FUNCTION_BLOCK XtsMover IMPLEMENTS I_Cyclic, I_XtsMover, I_Resettable, I_Object
VAR
	MyAxisRef : AXIS_REF;
	_MyAxisStatus : ST_AxisStatus;
	_MyNCData : NCTOPLC_AXIS_REF;
	TaskCollection : ObjectRunner<99>;
	EnableBehaviour : EnableDisableTask := (AxisRef := MyAxisRef);
	MoveBehaviour : MoveToPositionTask:= (AxisRef := MyAxisRef);
	HaltBehaviour : HaltMoverTask := (AxisRef := MyAxisRef);
	ResetBehaviour : CoEResetTask := (AxisRef := MyAxisRef);
	MoverActivateTrackBehaviour : ActivateTrackTask:= (AxisRef := MyAxisRef);
	_ipTcIoXtsMover	: I_TcIoXtsXpuMover;
	TrackChangeTrigger : R_TRIG;
	_MoverAbsMoveOptions : ST_MoveAbsoluteCAOptions;
	_stTmsActPositions : ST_PositionInfo;
	_CurrentTrack : I_XtsTrack;
	_myStatus : MoverStatus;
	_MyCAGroup : I_CollisionGroup;
	_ForwardOnly : BOOL := TRUE;
	myControllerOid: OTCID;
	MyId: UDINT;
	MoverID : T_MaxString;
	Initialised : BOOL;
	MyTrackCount : INT;
	MyTracks : ARRAY[0..MaxTracks] OF I_XtsTrack;
	NullTrack : XtsTrack('');
	_SetForce: LREAL;
	_SetCurrent: LREAL;
	_Gap : LREAL;
	_Acceleration : LREAL;
	_Deceleration : LREAL;
	_Jerk : LREAL;
	_DistanceDrivenInMM : LREAL;
	_AvoidingCollision: BOOL;
	_Mover1 : BOOL;
	myController: Tc3_XTS_Utility.I_McXtsMoverController;
END_VAR
VAR CONSTANT
	_MaxMoverVelocity : MC_LREAL := 4000.0;
	MaxTracks : INT := 5;
	InPositionToleranceForMoveChecks : LREAL := 0.001;
END_VAR

PROPERTY PUBLIC Acceleration : MC_LREAL
GET
Acceleration := MoveBehaviour.Acceleration;
END_GET
SET
MoveBehaviour.Acceleration := Acceleration;
_Acceleration := Acceleration;
END_SET
END_PROPERTY

METHOD ActivateTrack : HRESULT
VAR_INPUT
	Track : INT;
END_VAR
IF Track = 0 THEN
	ActivateTrack := -1;
	Base_Library.Tracing.Trace.Warning(MoverID, 'ActivateTrack Fail - Null Track');
	RETURN;
END_IF
IF MoverActivateTrackBehaviour.Busy THEN
	ActivateTrack := -2;
	Base_Library.Tracing.Trace.Warning(MoverID, 'ActivateTrack Fail - Activating');
	RETURN;
END_IF

IF NOT THIS^.IsStationary THEN
	ActivateTrack := -3;
	Base_Library.Tracing.Trace.Warning(MoverID, 'ActivateTrack Fail - Moving');
	RETURN;
END_IF

IF Track > MyTrackCount THEN
	ActivateTrack := -4;
	Base_Library.Tracing.Trace.Warning(MoverID, 'ActivateTrack Fail - Track not Registered');
	RETURN;
END_IF

IF MyTracks[Track - 1].MyOTCID = 0  THEN
	ActivateTrack := -5;
	Base_Library.Tracing.Trace.Warning(MoverID, 'ActivateTrack Fail - No Track');
	RETURN;
END_IF
	
Base_Library.Tracing.Trace.Verbose(MoverID, 'ActivateTrack Request Accepted');
MoverActivateTrackBehaviour.Execute(Track := MyTracks[Track - 1]);
_ipTcIoXtsMover.SetActiveTrackObjectId(nTrackObjectId := MyTracks[Track - 1].MyOTCID);
_CurrentTrack := MyTracks[Track - 1];
END_METHOD

METHOD ActivateZeroReferenceSystem : HRESULT
IF MoverActivateTrackBehaviour.Busy THEN
	ActivateZeroReferenceSystem := -1;
	Base_Library.Tracing.Trace.Warning(MoverID, 'ActivateZeroTrack Fail - Activating');
	RETURN;
END_IF
IF NOT THIS^.IsStationary THEN
	ActivateZeroReferenceSystem := -2;
	Base_Library.Tracing.Trace.Warning(MoverID, 'ActivateZeroTrack Fail - Moving');
	RETURN;
END_IF 

Base_Library.Tracing.Trace.Verbose(MoverID, 'ActivateTrack Request Accpeted');
MoverActivateTrackBehaviour.Execute(Track := NullTrack);
_CurrentTrack := 0;
END_METHOD

PROPERTY ActualForce : LREAL
GET
ActualForce := _SetForce;
END_GET
END_PROPERTY

PROPERTY ActualPosition : LREAL
GET
ActualPosition := MyAxisRef.NcToPlc.ActPos;
END_GET
END_PROPERTY

PROPERTY ActualTrackPosition : LREAL
GET
ActualTrackPosition := _stTmsActPositions.fTrackPosition;
END_GET
END_PROPERTY

PROPERTY ActualVelocity : LREAL
GET
ActualVelocity := MyAxisRef.NcToPlc.ActVelo;
END_GET
END_PROPERTY

PROPERTY AxisRef : Reference to Axis_ref
GET
AxisRef REF= MyAxisRef;
END_GET
END_PROPERTY

METHOD PUBLIC  Cycle : HRESULT
VAR_INPUT
END_VAR
IF Initialised THEN
	TaskCollection.Cycle();
	TrackChangeTrigger(CLK := MoverActivateTrackBehaviour.Done);
	IF TrackChangeTrigger.Q THEN
		_MoverAbsMoveOptions.PositionReferenceSystem :=  MoverActivateTrackBehaviour.NewTrackId;
		_MoverAbsMoveOptions.DynamicsReferenceSystem := MoverActivateTrackBehaviour.NewTrackId;
		MoveBehaviour.Options := _MoverAbsMoveOptions;	
	END_IF
	IF _ipTcIoXtsMover <> 0 THEN
		_stTmsActPositions := _ipTcIoXtsMover.GetPositionInfo();
		_SetForce := _ipTcIoXtsMover.GetSetForce();
		_SetCurrent := _ipTcIoXtsMover.GetSetCurrent();
		_myStatus.isMover1 := _ipTcIoXtsMover.GetIsMover1();
		_myStatus.isActive := _ipTcIoXtsMover.GetIsActive();
		_myStatus.isFrozen := _ipTcIoXtsMover.GetIsFrozen();
		_myStatus.isLost := _ipTcIoXtsMover.GetIsLost();
		_myStatus.isReadyForPositioning := _ipTcIoXtsMover.GetIsReadyForPositioning();
		_myStatus.hasControllerError := _ipTcIoXtsMover.GetMoverControllerError();
		_myStatus.driveState := _ipTcIoXtsMover.GetDriveStatus();
		_DistanceDrivenInMM := _ipTcIoXtsMover.GetDistanceDriven();
	END_IF
	_AvoidingCollision := MyAxisRef.NcToPlc.StateDWord2.Flags.AvoidingCollision;
ELSE
	Cycle := -1;
END_IF
MyAxisRef.ReadStatus();
_MyNCData := MyAxisRef.NcToPlc;
_MyAxisStatus := MyAxisRef.Status;
END_METHOD

PROPERTY PUBLIC Deceleration : MC_LREAL
GET
Deceleration := MoveBehaviour.Deceleration;
END_GET
SET
MoveBehaviour.Deceleration := Deceleration;
HaltBehaviour.Deceleration := Deceleration;
_Deceleration := Deceleration;
END_SET
END_PROPERTY

METHOD PUBLIC DisableMover : HRESULT
VAR_INPUT
END_VAR
IF NOT THIS^.IsEnabled THEN
	DisableMover := -1;
	Base_Library.Tracing.Trace.Warning(MoverID, 'Disable request Fail - Disabled'); 
	RETURN;
END_IF
	
Base_Library.Tracing.Trace.Verbose(MoverID, 'Disable Request Accepted');
EnableBehaviour.Disable();
END_METHOD

METHOD PUBLIC EnableMover : HRESULT
VAR_INPUT
END_VAR
IF EnableBehaviour.Busy THEN
	EnableMover := -1;
	Base_Library.Tracing.Trace.Warning(MoverID, 'Enable Request Failed - Enabling');
	RETURN;
END_IF
IF THIS^.IsEnabled THEN
	EnableMover := -2;
	Base_Library.Tracing.Trace.Warning(MoverID, 'Enable Request Failed - Enabled');
	RETURN;
END_IF
	
Base_Library.Tracing.Trace.Verbose(MoverID, 'Enable Request Accepted');
EnableBehaviour.Enable();
END_METHOD

PROPERTY ErrorID : UDINT
GET
ErrorID := _MyAxisStatus.ErrorID;
END_GET
END_PROPERTY

//FB_Init is always available implicitly and it is used primarily for initialization.
//The return value is not evaluated. For a specific influence, you can also declare the
//methods explicitly and provide additional code there with the standard initialization
//code. You can evaluate the return value.
METHOD FB_Init: BOOL
VAR_INPUT
    bInitRetains: BOOL; // TRUE: the retain variables are initialized (reset warm / reset cold)
    bInCopyCode: BOOL;  // TRUE: the instance will be copied to the copy code afterward (online change)   
END_VAR
TaskCollection.RegisterCyclic(EnableBehaviour);
TaskCollection.RegisterCyclic(ResetBehaviour);
TaskCollection.RegisterCyclic(HaltBehaviour);
TaskCollection.RegisterCyclic(MoveBehaviour);
TaskCollection.RegisterCyclic(MoverActivateTrackBehaviour);
END_METHOD

PROPERTY PUBLIC Gap : MC_LREAL
GET
Gap := MoveBehaviour.Gap;
END_GET
SET
IF Gap >= 50.0 THEN
	MoveBehaviour.Gap := Gap;
	HaltBehaviour.Gap := Gap;
	_Gap := Gap;
ELSE
	_Gap := 100.0;
	MoveBehaviour.Gap := 100.0;
	HaltBehaviour.Gap := 100.0;
END_IF
END_SET
END_PROPERTY

METHOD GetActiveTrackLength : LREAL
VAR_INPUT
END_VAR
GetActiveTrackLength := _CurrentTrack.TrackLength;
END_METHOD

METHOD GetMoverCtrlOTCID : XtsMoverControllerOTCID
VAR_INPUT
END_VAR
GetMoverCtrlOTCID := _ipTcIoXtsMover.GetMoverControllerOid();
END_METHOD

METHOD GetMoverOTCID : OTCID
VAR_INPUT
END_VAR
//GetMoverCtrlOTCID := _ipTcIoXtsMover.P_AxisOid;
END_METHOD

METHOD PUBLIC HaltAxis : HRESULT
VAR_INPUT
END_VAR
IF HaltBehaviour.Busy THEN
	HaltAxis := -1;
	Base_Library.Tracing.Trace.Warning(MoverID, 'Halt Request Fail - Halting');
	RETURN;
END_IF
	
Base_Library.Tracing.Trace.Verbose(MoverID, 'Halt Request Accepted');
HaltBehaviour.Execute();
END_METHOD

PROPERTY HasError : BOOL
GET
HasError := _MyAxisStatus.Error;
END_GET
END_PROPERTY

PROPERTY PUBLIC IdentInGroup : IDENT_IN_GROUP_REF
GET
IdentInGroup := UDINT_TO_IDENTINGROUP(id := _MyNCData.AxisId);
END_GET
END_PROPERTY

METHOD Initialise : HRESULT
VAR_INPUT
END_VAR
VAR
	i : INT;
END_VAR
IF Initialised THEN
	Initialise := -1;
	RETURN;
END_IF
IF _ipTcIoXtsMover = 0 THEN
	Initialise := -2;
	RETURN;
END_IF
IF NOT IsDetected THEN
	Initialise := -3;
	RETURN;
END_IF
IF MyTrackCount = 0 THEN
	Initialise := -4;
	RETURN;
END_IF
myController := _ipTcIoXtsMover.MoverController;
myControllerOid := _ipTcIoXtsMover.GetMoverControllerOid();
MyId := _ipTcIoXtsMover.P_AxisId;
MoverID := CONCAT('Mover ', TO_STRING(MyId));
_Mover1 := _ipTcIoXtsMover.GetIsMover1();
_CurrentTrack := MyTracks[MoversActiveTrack - 1];
Initialised := TRUE;
END_METHOD

PROPERTY IsActive : BOOL
GET
IsActive := _myStatus.isActive;
END_GET
END_PROPERTY

PROPERTY IsAMover1 : BOOL
GET
IsAMover1 := _Mover1;
END_GET
END_PROPERTY

PROPERTY IsAvoidingCollision : BOOL
GET
isAvoidingCollision := _AvoidingCollision;
END_GET
END_PROPERTY

PROPERTY IsDetected : BOOL
GET
IsDetected := MyAxisRef.NcToPlc.AxisId <> 0;
END_GET
END_PROPERTY

PROPERTY IsEnabled : BOOL
GET
IsEnabled :=  NOT _MyAxisStatus.Disabled;
END_GET
END_PROPERTY

PROPERTY IsStationary : BOOL
GET
IsStationary := _MyAxisStatus.NotMoving;
END_GET
END_PROPERTY

PROPERTY PUBLIC Jerk : MC_LREAL
GET
Jerk := MoveBehaviour.Jerk;
END_GET
SET
MoveBehaviour.Jerk := Jerk;
HaltBehaviour.Jerk := Jerk;
_Jerk := Jerk;
END_SET
END_PROPERTY

PROPERTY PUBLIC MoversActiveTrack : INT
GET
VAR
	i : INT;
END_VAR
FOR i := 0 TO MyTrackCount - 1 DO
	IF MyTracks[i].MyOTCID =  _ipTcIoXtsMover.GetActiveTrackObjectId() THEN
		MoversActiveTrack := i + 1;
		EXIT;
	END_IF
END_FOR
END_GET
END_PROPERTY

PROPERTY PUBLIC MoverXtsIoEnvInterface : I_TcIoXtsXpuMover
GET
MoverXtsIoEnvInterface := _ipTcIoXtsMover;
END_GET
SET
_ipTcIoXtsMover := MoverXtsIoEnvInterface;
END_SET
END_PROPERTY

METHOD PUBLIC MoveTo : HRESULT
VAR_INPUT
	RequiredPosition : MC_LREAL;
	MoveVelocity : MC_LREAL;
	NonModuloMove : BOOL;
END_VAR
IF MoveBehaviour.Busy THEN
	Base_Library.Tracing.Trace.Warning(MoverID, 'Mover Called While Busy');
	MoveTo := -1;
	RETURN;
END_IF
IF MoveVelocity > _MaxMoverVelocity THEN
	Base_Library.Tracing.Trace.Warning(MoverID, 'Move Velo Too High');
	MoveTo := -2;
	RETURN;
END_IF
IF MoveVelocity <= 0.0 THEN
	Base_Library.Tracing.Trace.Warning(MoverID, 'Move Velo Less Than Zero');
	MoveTo := -3;
	RETURN;
END_IF
IF Gap <= 50.0 THEN
	Base_Library.Tracing.Trace.Warning(MoverID, 'Move Gasp Too Small');
	MoveTo := -4;
	RETURN;
END_IF

Base_Library.Tracing.Trace.Verbose(moverID, concat('Move Accepted to : ',TO_STRING(RequiredPosition)));

IF NonModuloMove THEN
	THIS^.MoveBehaviour.MoveTo(Position := RequiredPosition, 
									Velocity := MoveVelocity, 
									Direction := Tc3_Mc3Definitions.MC_DIRECTION.mcDirectionNonModulo, 
									Turns := 0);
	MoveTo := 1;
END_IF

IF NOT NonModuloMove AND _ForwardOnly THEN
	MoveTo := THIS^.MoveBehaviour.MoveTo(Position := RequiredPosition, 
									Velocity := MoveVelocity, 
									Direction := Tc3_Mc3Definitions.MC_DIRECTION.mcDirectionPositive, 
									Turns := 0);
	MoveTo := 2;
END_IF

IF NOT NonModuloMove AND NOT _ForwardOnly THEN
	IF RequiredPosition > MyAxisRef.NcToPlc.ModuloActPos THEN
		MoveTo := THIS^.MoveBehaviour.MoveTo(Position := RequiredPosition, 
									Velocity := MoveVelocity, 
									Direction := Tc3_Mc3Definitions.MC_DIRECTION.mcDirectionPositive, 
									Turns := 0);
		MoveTo := 3;
	ELSE
		MoveTo := THIS^.MoveBehaviour.MoveTo(Position := RequiredPosition, 
									Velocity := MoveVelocity, 
									Direction := Tc3_Mc3Definitions.MC_DIRECTION.mcDirectionNegative, 
									Turns := 0);
		MoveTo := 4;
	END_IF
END_IF
END_METHOD

PROPERTY MyCAGroup : I_CollisionGroup
GET
MyCAGroup := _MyCAGroup;
END_GET
SET
_MyCAGroup := MyCAGroup;
END_SET
END_PROPERTY

PROPERTY PositiveDirectionOnly : BOOL
GET
PositiveDirectionOnly := _ForwardOnly;
END_GET
SET
_ForwardOnly := PositiveDirectionOnly;
END_SET
END_PROPERTY

METHOD RegisterTracks : HRESULT
VAR_INPUT
	Track : I_XtsTrack;
END_VAR
VAR
	Registered : BOOL;
	i : INT;
END_VAR
IF Track = 0 THEN
	RegisterTracks := -1;
	RETURN;
END_IF
Registered := FALSE;
FOR i := 0 TO 5 DO 
	IF Track = MyTracks[i] THEN
		Registered := TRUE;
	END_IF
END_FOR
IF Registered THEN
	RegisterTracks := -2;
	RETURN;
END_IF
FOR i := 0 TO 5 DO
	IF MyTracks[i] = 0 THEN
		MyTracks[i] := Track;
		MyTrackCount := MyTrackCount + 1;
		EXIT;
	END_IF
END_FOR
END_METHOD

METHOD RegisterWithParent
VAR_INPUT
	Parent	: I_HostObjects;
END_VAR
Parent.RegisterCyclic(THIS^);
END_METHOD

METHOD PUBLIC Reset : HRESULT
VAR_INPUT
END_VAR
IF ResetBehaviour.Busy THEN
	Base_Library.Tracing.Trace.Warning(MoverID, 'Reset Request Failed - Reseting');
	Reset := -1;
	RETURN;
END_IF
 
IF NOT (_MyAxisStatus.Error OR _MyAxisStatus.NotMoving) THEN
	Base_Library.Tracing.Trace.Warning(MoverID, 'Reset Request Failed - Not Allowed');
	Reset := -2;
	RETURN;
END_IF

Base_Library.Tracing.Trace.Verbose(MoverID, 'Reset Request Accepted');
ResetBehaviour.Reset();
MoveBehaviour.Abort();
END_METHOD

METHOD SetForceCouple : HRESULT
VAR_INPUT
	XtsMoverCtrlOTCID : Tc3_XTS_Utility.XtsMoverControllerOTCID;
END_VAR
IF _ipTcIoXtsMover = 0 THEN
	SetForceCouple := - 1;
	RETURN;
END_IF

_ipTcIoXtsMover.MoverController.SetForceCouple(nForceCouple := XtsMoverCtrlOTCID);
END_METHOD

METHOD SetMoverActiveTrack : HRESULT
VAR_INPUT
	Track : INT;
END_VAR
IF Track = 0 THEN
	SetMoverActiveTrack := -1;
	RETURN;
END_IF

IF NOT THIS^.IsStationary THEN
	SetMoverActiveTrack := -3;
	RETURN;
END_IF

IF Track > MyTrackCount THEN
	SetMoverActiveTrack := -4;
	RETURN;
END_IF

IF MyTracks[Track - 1].MyOTCID = 0  THEN
	SetMoverActiveTrack := -5;
	RETURN;
END_IF
	
_ipTcIoXtsMover.SetActiveTrackObjectId(nTrackObjectId := MyTracks[Track - 1].MyOTCID);
_CurrentTrack := MyTracks[Track - 1];
END_METHOD

METHOD SetParameterSet : HRESULT
VAR_INPUT
	ParameterSet : OTCID;
END_VAR
IF ParameterSet = 0 THEN
	RETURN;
	SetParameterSet := -1;
END_IF

myController.SetDefaultParameterSet(ParameterSet);
END_METHOD

METHOD SetSimDetectionPartAndPosition : BOOL
VAR_INPUT
	Part : OTCID;
	Position : LREAL;
END_VAR
_ipTcIoXtsMover.SetSimulatedStartUpPart(Part);
_ipTcIoXtsMover.SetSimulatedStartUpPosition(Position);
END_METHOD

METHOD SwapMover : HRESULT
VAR_INPUT
    MoverToSwapWith : MoverOTCID;
END_VAR
_ipTcIoXtsMover.swapmover(nSwapMoverObjectId := MoverToSwapWith);
END_METHOD

METHOD TriggerMoverArrive : HRESULT
VAR_INPUT
END_VAR
IF _ipTcIoXtsMover = 0 THEN
	TriggerMoverArrive := - 1;
	RETURN;
END_IF
IF _myStatus.isActive THEN
	TriggerMoverArrive := - 2;
	RETURN;
END_IF

_ipTcIoXtsMover.TriggerArrive();
END_METHOD

METHOD TriggerMoverLeave : HRESULT
VAR_INPUT
END_VAR
IF _ipTcIoXtsMover = 0 THEN
	TriggerMoverLeave := -1;
	RETURN;
END_IF
IF NOT _myStatus.isActive THEN
	TriggerMoverLeave := -2;
	RETURN;
END_IF
IF NOT IsStationary THEN
	TriggerMoverLeave := -3;
	RETURN;
END_IF

_ipTcIoXtsMover.TriggerLeave();
END_METHOD

END_FUNCTION_BLOCK

(* stored: Version 1.1.0.1
   POU XtsMover: Id {f9a43ed2-0578-4aed-857c-1a3adef0c7f6}, SpecialFunc None
   Folder Administration: Id {660864df-8996-42d7-8e95-bfca1c90696e}
   Folder Commands: Id {db0a893b-cc1a-482e-a432-7e9d568c5112}
   Folder Dynamics: Id {6b49cc7a-c913-475a-9f9a-db91d65d07e1}
   Folder ICyclic: Id {895ad701-1670-4c6d-921e-cd7ccab0c12a}
   Folder Status: Id {b27ba391-8a3b-4e51-ae24-bae43a7b6e5f}
   Property Acceleration: Id {5cd04126-8ceb-4f9d-a4c5-c87e7e11d0e6}
   Get Get: Id {89c9e6d0-5dfa-4531-97de-32e16eb2e196}
   Set Set: Id {95cc2e62-d911-4757-83d0-b9b38a36fdde}
   Method ActivateTrack: Id {f7604675-5338-4e11-9132-b17d5df72cc8}
   Method ActivateZeroReferenceSystem: Id {f593e12a-c440-483d-8309-49c5dc48d5f1}
   Property ActualForce: Id {1098aa35-8fe0-43b3-b10d-2dbf741e0cc6}
   Get Get: Id {10e9735a-f2ce-4d5a-ac32-880505647b0c}
   Property ActualPosition: Id {97d35bbc-7d79-4ab6-acbe-efd9e040cf7e}
   Get Get: Id {e195bcb1-e534-4753-a471-130b7260a030}
   Property ActualTrackPosition: Id {f0eba487-b575-4c34-b1c8-92f6f0d4e9ff}
   Get Get: Id {12465534-ac82-4003-9fc9-808736ed6478}
   Property ActualVelocity: Id {464c1699-07a2-4876-88f8-424d8c881d6d}
   Get Get: Id {cf005a5e-7c46-4435-9144-c308d46bca18}
   Property AxisRef: Id {a7d5ea1d-51bb-4c87-90b3-db66fd196d20}
   Get Get: Id {8c3b00e4-86fb-42e3-b0e0-5789e5045419}
   Method Cycle: Id {b5956233-12ba-4cb8-805f-5693aec42bed}
   Property Deceleration: Id {3def2bbc-f7ec-4120-acb9-2ff2a2789bd5}
   Get Get: Id {e6097884-8279-4e20-92f9-6fb8b5120af4}
   Set Set: Id {dbf3cf03-c8db-40c9-ab3e-669bb5cdced1}
   Method DisableMover: Id {a82f95fa-77b4-4c5e-ae67-686dbd3b2d8d}
   Method EnableMover: Id {d130fe63-f34a-4455-8bb8-4dfcc482e573}
   Property ErrorID: Id {b75590a2-f278-4019-b919-db0f4a472676}
   Get Get: Id {b4aa86dd-bc0f-49f0-ac26-dce353b288a4}
   Method FB_Init: Id {e6cdc000-5fb3-42ba-8ce8-01408a72b06f}
   Property Gap: Id {dd72da9d-fc94-421a-8ee7-a84a721dd20c}
   Get Get: Id {5c8fd02d-70e7-4f46-b386-6000a46a3487}
   Set Set: Id {280f9258-e1cd-43be-bf57-16929cbbc8d6}
   Method GetActiveTrackLength: Id {4b840da8-e3cc-46e4-bf3c-0fcb89870f67}
   Method GetMoverCtrlOTCID: Id {6852d0c0-13fb-4a6d-9e8b-5d538e770d2f}
   Method GetMoverOTCID: Id {0ee3ade7-076c-46ec-8833-0ad2fc45f400}
   Method HaltAxis: Id {b177db81-8e99-498a-a7a2-cd0938dd7a2c}
   Property HasError: Id {20bfb091-3a51-46b6-b1c3-86998c1edac5}
   Get Get: Id {d8e26ea2-dd1a-4fc5-8d5e-87f1bef9cf9c}
   Property IdentInGroup: Id {4d5563a0-634a-4074-a0e4-612875dd790c}
   Get Get: Id {6419a53d-e416-464a-881c-e300db0a9add}
   Method Initialise: Id {158eaadb-7779-40c3-b4d7-ef64750e6b36}
   Property IsActive: Id {382be57c-1eca-4414-86e7-197f5c6f4f45}
   Get Get: Id {ea8b86db-8f1a-4f2a-bfa5-c492ca87a414}
   Property IsAMover1: Id {028ba926-1842-41e8-aa1c-c4ef6eef97c2}
   Get Get: Id {4143db0b-f9d6-45f3-9ff5-3b331e0fc8b8}
   Property IsAvoidingCollision: Id {da7886a8-9c9c-4ae2-bbae-548351ceb9d3}
   Get Get: Id {07cfba67-3f84-4db0-a72d-fbe6f6b78e00}
   Property IsDetected: Id {be1fef7b-c667-4190-a068-7a115721883c}
   Get Get: Id {48fddea6-2ee5-46a7-89af-2a78eb812316}
   Property IsEnabled: Id {8e71c4a3-2ef0-42bd-bfd7-77e344d1bd40}
   Get Get: Id {5b5f088a-6649-46f8-bd13-7cd57e7cee10}
   Property IsStationary: Id {7f9079b5-4633-4e28-a842-9024cc33e246}
   Get Get: Id {f4fdfa27-6cb9-47cc-bbad-29d2dbcc8306}
   Property Jerk: Id {fbc5f504-aa6b-48f8-8a62-bbde3b74b20e}
   Get Get: Id {98c0c9db-aae6-4788-a223-2bf5fa007418}
   Set Set: Id {6a6a16a3-4f19-4f4d-bd8d-8441ae3b5cf2}
   Property MoversActiveTrack: Id {15471ba0-8341-48c7-a2d0-01ca6286078a}
   Get Get: Id {2721855b-e1d8-4f74-a352-28794ee4ae69}
   Property MoverXtsIoEnvInterface: Id {6aaf98f4-e1bc-4f35-afbe-48664404e767}
   Get Get: Id {5b75808a-7c24-4c09-8809-4a555d5acdb1}
   Set Set: Id {57119448-dfbf-405e-ade1-72aad5224720}
   Method MoveTo: Id {ea6488b0-fefd-4f9f-a3b2-cfd8c6f64d05}
   Property MyCAGroup: Id {ef4ebc28-e3bd-4e4a-8472-4104ad14ebae}
   Get Get: Id {d4b3e253-6981-43ac-859c-776f6b4fec7d}
   Set Set: Id {54c77228-8f9c-4310-9bfc-ef466b7143ba}
   Property PositiveDirectionOnly: Id {993fe16b-05a5-4eca-a38c-6463f3e7295c}
   Get Get: Id {581a1e54-141a-440c-9d85-39be9d6e8e36}
   Set Set: Id {aede2ad8-809d-4697-b667-b49152253954}
   Method RegisterTracks: Id {33623a4f-6a2b-45ed-b81c-64a295cf1295}
   Method RegisterWithParent: Id {0c8fc6cb-d807-4926-a588-870aa525c7f2}
   Method Reset: Id {e9d8249c-2f88-4980-a483-ceda82c7ab80}
   Method SetForceCouple: Id {655fe1cd-78c7-4097-b5c7-b05e68cd5f7e}
   Method SetMoverActiveTrack: Id {d6a4b78b-2758-4ca3-91dd-004aef96a776}
   Method SetParameterSet: Id {a2d3312c-642a-4ded-95b4-a250a99284ac}
   Method SetSimDetectionPartAndPosition: Id {7c9e452d-fc91-446a-83ce-0915a34e15cf}
   Method SwapMover: Id {075d081f-a4ad-470f-95aa-ced1f28cc5a8}
   Method TriggerMoverArrive: Id {9bb7f072-ab21-4ec2-9434-ad1366cf5fb7}
   Method TriggerMoverLeave: Id {074e60e5-1df3-46d8-92fd-930fc05fcb13} *)
